INTERFACE I_AnalogScalable EXTENDS I_Base

PROPERTY Scale : I_AnalogScale
GET
END_GET
SET
END_SET
END_PROPERTY

END_INTERFACE

(* stored: Version 1.1.0.1, ProductVersion 3.1.4026.18
   Itf I_AnalogScalable: Id {62c21804-74ca-483e-b7ff-e9198c37548f}
   Property Scale: Id {09264835-234c-4f51-aa87-d67af919eab0}
   Get Get: Id {a087bf11-d4fd-49f8-8c08-35b444c8ec03}
   Set Set: Id {38f8c6cf-4c01-4b06-a56c-92475cb2c7ff} *)
